// TIA Portal V19 export
TYPE "LAF_typeDriveDiagInterfaceHmi"
TITLE = LAF_typeDriveDiagStatus
// HMI interface structure for drive diagnostic
// stored: Access Published
   STRUCT
      hmi : "LAF_typeHmiDiagData";
      axis : "LAF_typeAxisDiagData";
      sina : "LAF_typeSinaDiagData";
   END_STRUCT;
END_TYPE
